// TIA Portal V17 export
// export: Created 2025-05-22T06:00:57.2159887Z, ExportSetting WithDefaults, DisplayName Totally Integrated Automation Portal, DisplayVersion V17 Update 8, DisplayName TIA Portal Openness, DisplayVersion V17 Update 8, DisplayName TIA Portal Version Control Interface, DisplayVersion V17, DisplayName SINAMICS Startdrive Advanced, DisplayVersion V17 SP2, DisplayName SINAMICS Startdrive G110M, G120, G120C, G120D, G120P, G115D, DisplayVersion V17 SP2, DisplayName SINAMICS Startdrive G130, G150, S120, S150, SINAMICS MV, S210, DisplayVersion V17 SP2, DisplayName STEP 7 Professional, DisplayVersion V17 Update 8, DisplayName SINUMERIK ONE STEP 7 Toolbox, DisplayVersion V17 Update 12, DisplayName SINUMERIK ONE PLC Basic Program Plus, DisplayVersion V17 Update 12, DisplayName SINUMERIK 840D sl STEP 7 Toolbox, DisplayVersion V17 Update 12, DisplayName STEP 7 Safety, DisplayVersion V17 Update 6, DisplayName WinCC Advanced, DisplayVersion V17 Update 8
DATA_BLOCK "DB3500_UNIT_2_FIXTURE_1"   // DB3500
{ DB_Accessible_From_OPC_UA := 'FALSE' }
VERSION : 0.1
// stored: AutoNumber false, DBAccessibleFromOPCUA false, DBAccessibleFromWebserver true, InstanceOfName FB2500_FIXTURE_CLADDING, InstanceOfType FB
"FB2500_FIXTURE_CLADDING"
   // VAR_INPUT
   //    PART_PRESENT_FACE_SENSOR : Bool;
   //    PART_STATUS_PRESENT : Bool;
   //    PART_STATUS_VIRTUAL_PART : Bool;
   //    PART_STATUS_MASTER_PART : Bool;
   //    STATION_PART_PRESENT : Bool;
   //    STATION_NO_PART : Bool;
   //    STATION_PART_HAT_POSITION : Bool;
   //    STATION_PART_CLAMPED : Bool;
   //    STATION_PART_UNCLAMPED : Bool;
   //    STATION_CLAMPED_WITHOUT_PART : Bool;
   //    VERIFY_FIXTURE_CLAMPED : Bool;
   //    GRIPPER_CLOSE : Bool;
   //    GRIPPER_OPEN : Bool;
   //    GRIPPER_CLOSED : Bool;
   //    "GRIPPER OPENED" : Bool;
   //    M_FIXTURE_GRIPPER_CLOSE : Bool;
   //    M_FIXTURE_GRIPPER_OPEN : Bool;
   //    UP_SEALING_STRUCTURE_CLOSED : Bool;
   //    DOWN_SEALING_STRUCTURE_CLOSED : Bool;
   //    PART_TYPE_FIXTURES : Bool;
   //    ROBOT_PART_LOAD_UNLOAD : Bool;
   //    ROBOT_OUT_OF_COLLISION : Bool;
   //    E_AXIS_HOME_POS : Bool;
   //    W_AXIS_CLAMP_CHECK_POS : Bool;
   //    W_AXIS_UNCLAMP_CHECK_POS : Bool;
   //    UNIT_NO : UInt;
   //    FIXTURE_NO : UInt;
   // END_VAR
   // VAR_OUTPUT
   //    NOT_CLAMPED_DURING_MACHINING_A : Bool;
   //    PART_PRESENT_DISCORDANCY_A : Bool;
   //    PART_TYPE_DISCORDANCY_A : Bool;
   //    PART_TYPE_ORIENTATED_DISCORDANCY_A : Bool;
   // END_VAR
   // VAR RETAIN
   //    DATA : "FIXTURE_STATUS";
   // END_VAR
BEGIN
END_DATA_BLOCK
